Staubli VAL3: Welcome.pgx

program Welcome()
begin

  call UI:Form_Welcome("激光软件LasMAN3.7",bWelcome)




end
